SYSTEM Test Big Computation par 40
  (* Version 1.0, 2005-12-19, Goran Cengic, Chalmers *)
  DEVICE Test Device : DeviceType_not_used
    RESOURCE Test Resource : ResourceType_not_used
      FBS
        restart : E_RESTART;
        stop : E_STOP;
        split : E_SPLIT40;
        big1 : BigComputation;
        big2 : BigComputation;
        big3 : BigComputation;
        big4 : BigComputation;
        big5 : BigComputation;
        big6 : BigComputation;
        big7 : BigComputation;
        big8 : BigComputation;
        big9 : BigComputation;
        big10 : BigComputation;
        big11 : BigComputation;
        big12 : BigComputation;
        big13 : BigComputation;
        big14 : BigComputation;
        big15 : BigComputation;
        big16 : BigComputation;
        big17 : BigComputation;
        big18 : BigComputation;
        big19 : BigComputation;
        big20 : BigComputation;
        big21 : BigComputation;
        big22 : BigComputation;
        big23 : BigComputation;
        big24 : BigComputation;
        big25 : BigComputation;
        big26 : BigComputation;
        big27 : BigComputation;
        big28 : BigComputation;
        big29 : BigComputation;
        big30 : BigComputation;
        big31 : BigComputation;
        big32 : BigComputation;
        big33 : BigComputation;
        big34 : BigComputation;
        big35 : BigComputation;
        big36 : BigComputation;
        big37 : BigComputation;
        big38 : BigComputation;
        big39 : BigComputation;
        big40 : BigComputation;
      END_FBS
      EVENT_CONNECTIONS
        restart.COLD TO split.EI;
        split.EO1 TO big1.EI;
        split.EO2 TO big2.EI;
        split.EO3 TO big3.EI;
        split.EO4 TO big4.EI;
        split.EO5 TO big5.EI;
        split.EO6 TO big6.EI;
        split.EO7 TO big7.EI;
        split.EO8 TO big8.EI;
        split.EO9 TO big9.EI;
        split.EO10 TO big10.EI;
        split.EO11 TO big11.EI;
        split.EO12 TO big12.EI;
        split.EO13 TO big13.EI;
        split.EO14 TO big14.EI;
        split.EO15 TO big15.EI;
        split.EO16 TO big16.EI;
        split.EO17 TO big17.EI;
        split.EO18 TO big18.EI;
        split.EO19 TO big19.EI;
        split.EO20 TO big20.EI;
        split.EO21 TO big21.EI;
        split.EO22 TO big22.EI;
        split.EO23 TO big23.EI;
        split.EO24 TO big24.EI;
        split.EO25 TO big25.EI;
        split.EO26 TO big26.EI;
        split.EO27 TO big27.EI;
        split.EO28 TO big28.EI;
        split.EO29 TO big29.EI;
        split.EO30 TO big30.EI;
        split.EO31 TO big31.EI;
        split.EO32 TO big32.EI;
        split.EO33 TO big33.EI;
        split.EO34 TO big34.EI;
        split.EO35 TO big35.EI;
        split.EO36 TO big36.EI;
        split.EO37 TO big37.EI;
        split.EO38 TO big38.EI;
        split.EO39 TO big39.EI;
        split.EO40 TO big40.EI;
        big40.EO TO stop.STOP;
      END_CONNECTIONS
    END_RESOURCE
  END_DEVICE
END_SYSTEM
